PROGRAM PRG_1_PlcTask
VAR
END_VAR


PRG_2_PMPS();
PRG_3_LOG();
PRG_Diffractometer();
PRG_LAS();
PRG_SDS();
PRG_RotDet();
//PRG_Questar();
PRG_SpetrometerArm();
PRG_SSL();
PRG_Cryo();

END_PROGRAM

(* stored: Version 1.1.0.1, ProductVersion 3.1.4022.18
   POU PRG_1_PlcTask: Id {ffe71f0c-bf77-4cce-b8e1-24b1bdf50732}, SpecialFunc None *)
